// TIA Portal V16 export
// export: Created 2024-06-24T15:42:27.3705035Z, ExportSetting WithDefaults, DisplayName Totally Integrated Automation Portal, DisplayVersion V16, DisplayName TIA Portal Version Control Interface, DisplayVersion V16, DisplayName TIA Portal Openness, DisplayVersion V16, DisplayName STEP 7 Professional, DisplayVersion V16, DisplayName STEP 7 Safety, DisplayVersion V16, DisplayName WinCC Advanced, DisplayVersion V16
FUNCTION_BLOCK "FB_Pusher"   // FB1, LAD
{ S7_Optimized_Access := 'TRUE' }
VERSION : 0.1
// stored: AutoNumber true, IsIECCheckEnabled false, IsRetainMemResEnabled false, MemoryReserve 100, SetENOAutomatically false, UDAEnableTagReadback false
   VAR_INPUT
      "machine ready" : Bool;
      "front limit" : Bool;
      "back limit" : Bool;
   END_VAR
   VAR_OUTPUT
      extend : Bool;
      "counter" : Bool;
   END_VAR
   VAR_IN_OUT
      start : Bool;
      done : Bool;
   END_VAR
   VAR
      "step" : Array[0..19] of Bool;
   END_VAR
   VAR_TEMP   // added for the SCL form of the ladder/FBD networks
      _w1 : Bool;
   END_VAR
BEGIN

REGION Network 1
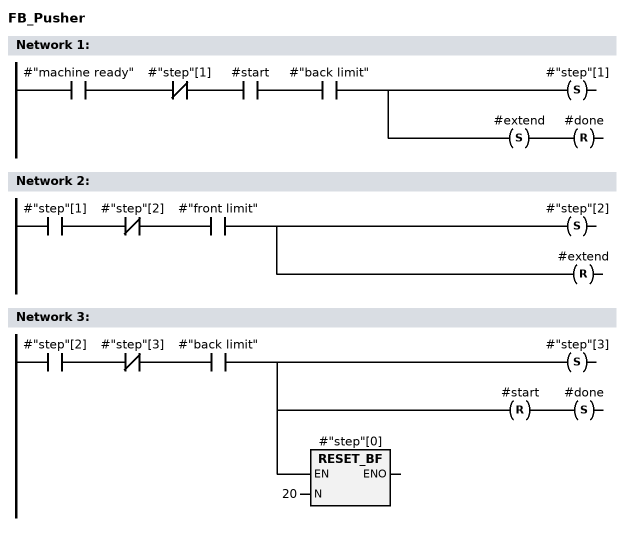
   RUNG wire#powerrail
      Contact( #"machine ready" )
      I_Contact( #"step"[1] )
      Contact( #start )
      Contact( #"back limit" )
      wire#w1
      S_Coil( #"step"[1] )
   END_RUNG
   RUNG wire#w1
      S_Coil( #extend )
      R_Coil( #done )
   END_RUNG
   // the same network as SCL:
   #_w1 := #"machine ready" AND NOT #"step"[1] AND #start AND #"back limit";
   IF #_w1 THEN
       #"step"[1] := TRUE;
       #extend := TRUE;
       #done := FALSE;
   END_IF;
END_REGION

REGION Network 2
   RUNG wire#powerrail
      Contact( #"step"[1] )
      I_Contact( #"step"[2] )
      Contact( #"front limit" )
      wire#w1
      S_Coil( #"step"[2] )
   END_RUNG
   RUNG wire#w1
      R_Coil( #extend )
   END_RUNG
   // the same network as SCL:
   #_w1 := #"step"[1] AND NOT #"step"[2] AND #"front limit";
   IF #_w1 THEN
       #"step"[2] := TRUE;
       #extend := FALSE;
   END_IF;
END_REGION

REGION Network 3
   // no SCL statement known for RBitfield: written as a call
   #_w1 := #"step"[2] AND NOT #"step"[3] AND #"back limit";
   IF #_w1 THEN
       #"step"[3] := TRUE;
       #start := FALSE;
       #done := TRUE;
       RESET_BF(operand := #"step"[0], n := 20);
   END_IF;
END_REGION
END_FUNCTION_BLOCK
